TYPE E_DisconnectorStatus :
(
    READY := 0,          // Hazır
    OPERATING := 1,      // Hareket halinde
    INTERLOCKED := 2,    // Interlock aktif
    FAULTED := 3,        // Arızalı
    NO_CONTROL := 4,     // PLC kontrol yok
    MAINTENANCE := 5     // Bakım gerekli
);
END_TYPE

(* stored: Version 1.1.0.1, ProductVersion 3.1.4024.15
   EnumerationTextList E_DisconnectorStatus: Id {80a2e924-4548-4f90-b390-25150b17e4e6} *)
